PROGRAM MAIN
VAR
	
IN_TEST_1 AT%I* : BOOL;
		
END_VAR

END_PROGRAM

(* stored: Version 1.1.0.1, ProductVersion 3.1.4024.9
   POU MAIN: Id {28c6f53e-9ffe-4339-a37a-f92f28e532a1}, SpecialFunc None *)
